PROGRAM ActuationSystems
VAR
fbMainJibCylinder : ValveControlledCylinder;
fbKnuckleJibCylinder : ValveControlledCylinder;
fbHPU : HPU;
END_VAR

fbHPU(
);

fbMainJibCylinder(
ReturnPressure := G_ActuationSystems.ReturnPressure,
SupplyPressure := G_ActuationSystems.SupplyPressure,
par := Param.pMainJibCylinder
);

fbKnuckleJibCylinder(
ReturnPressure := G_ActuationSystems.ReturnPressure,
SupplyPressure := G_ActuationSystems.SupplyPressure,
par := Param.pMainKnuckleCylinder
);

END_PROGRAM

(* stored: Version 1.1.0.1, ProductVersion 3.1.4024.9
   POU ActuationSystems: Id {3cabdd9c-217f-443b-9923-404fabc5dbf5}, SpecialFunc None *)
